Staubli VAL3: decTrajPtCartesian.pgx

public program decTrajPtCartesian(bool& x_bFlag)
  local num l_nIndex
  local num l_nRetVal
begin
  // decode message ID 31 body (data)

  // assume failure to decode
  rosTrajPtCartesianAck.header.nReplyCode=2

  // sequence
  l_nRetVal=fromBinary(rosTrajPtCartesianMsg.body.nData,4,"-4l",rosTrajPtCartesianMsg.cartesianTrajPt.nSeq)
  if(l_nRetVal!=1)
    x_bFlag=false
    return
  endIf

  // position[3]
  for l_nIndex=0 to 2 step 1
    l_nRetVal=fromBinary(rosTrajPtCartesianMsg.body.nData[(l_nIndex*4)+4],4,"4.0l",rosTrajPtCartesianMsg.cartesianTrajPt.nPosition[l_nIndex])
    if(l_nRetVal!=1)
      x_bFlag=false
      return
    endIf
  endFor

  // orientation[4]
  for l_nIndex=0 to 3 step 1
    l_nRetVal=fromBinary(rosTrajPtCartesianMsg.body.nData[(l_nIndex*4)+16],4,"4.0l",rosTrajPtCartesianMsg.cartesianTrajPt.nOrientation[l_nIndex])
    if(l_nRetVal!=1)
      x_bFlag=false
      return
    endIf
  endFor

  // velocity
  l_nRetVal=fromBinary(rosTrajPtCartesianMsg.body.nData[32],4,"4.0l",rosTrajPtCartesianMsg.cartesianTrajPt.nVelocity)
  if(l_nRetVal!=1)
    x_bFlag=false
    return
  endIf

  // acceleration
  l_nRetVal=fromBinary(rosTrajPtCartesianMsg.body.nData[36],4,"4.0l",rosTrajPtCartesianMsg.cartesianTrajPt.nAcceleration)
  if(l_nRetVal!=1)
    x_bFlag=false
    return
  endIf

  // blending radius
  l_nRetVal=fromBinary(rosTrajPtCartesianMsg.body.nData[40],4,"4.0l",rosTrajPtCartesianMsg.cartesianTrajPt.nBlendingRadius)
  if(l_nRetVal!=1)
    x_bFlag=false
    return
  endIf

  // duration
  l_nRetVal=fromBinary(rosTrajPtCartesianMsg.body.nData[44],4,"4.0l",rosTrajPtCartesianMsg.cartesianTrajPt.nDuration)
  if(l_nRetVal!=1)
    x_bFlag=false
    return
  endIf

  // decoding successful
  rosTrajPtCartesianAck.header.nReplyCode=1
  rosTrajPtCartesianAck.cartesianTrajPt.nSeq=rosTrajPtCartesianMsg.cartesianTrajPt.nSeq
  x_bFlag=true
end
